       J1 = 0.0 deg, J2 = 0.0 deg
 };
P[142] {
    GP1:
        UF : 6, UT : 5,     CONFIG: 'N U T, 0, 0, 0',
       X = -379.5 mm, Y = 409.2 mm, Z = 657.7 mm,
       W = -12.0 deg, P = 10.7 deg,
    GP2:
        UF : 1, UT : 2,
       J1 = 0.0 deg, J2 = 0.0 deg
 };
P[387] {
    GP1:
        UF : 6, UT : 5,     CONFIG: 'N U T, 0, 0, 0',
 X = -362.5 mm, Y = 480.2 mm, Z = 657.7 mm,       W = -12.0 deg, P = 10.7 deg,
    GP2:
        UF : 1, UT : 2,
       J1 = 0.0 deg, J2 = 0.0 deg
 };
P[143] {
    GP1:
        UF : 6, UT : 5,     CONFIG: 'N U T, 0, 0, 0',
       X = -383.8 mm, Y = 412.9 mm, Z = 657.7 mm,
       W = -11.8 deg, P = 10.5 deg,
    GP2:
        UF : 1, UT : 2,
       J1 = 0.0 deg, J2 = 0.0 deg
 };
P[388] {
    GP1:
        UF : 6, UT : 5,     CONFIG: 'N U T, 0, 0, 0',
 X = -366.8 mm, Y = 483.9 mm, Z = 657.7 mm,       W = -11.8 deg, P = 10.5 deg,
    GP2:
        UF : 1, UT : 2,
       J1 = 0.0 deg, J2 = 0.0 deg
 };
P[144] {
    GP1:
        UF : 6, UT : 5,     CONFIG: 'N U T, 0, 0, 0',
       X = -385.4 mm, Y = 414.3 mm, Z = 657.7 mm,
       W = -12.1 deg, P = 10.1 deg,
    GP2:
        UF : 1, UT : 2,
       J1 = 0.0 deg, J2 = 0.0 deg
 };
P[389] {
    GP1:
        UF : 6, UT : 5,     CONFIG: 'N U T, 0, 0, 0',
 X = -368.4 mm, Y = 485.3 mm, Z = 657.7 mm,       W = -12.1 deg, P = 10.1 deg,
    GP2:
        UF : 1, UT : 2,
       J1 = 0.0 deg, J2 = 0.0 deg
 };
P[145] {
    GP1:
        UF : 6, UT : 5,     CONFIG: 'N U T, 0, 0, 0',
       X = -393.1 mm, Y = 420.6 mm, Z = 657.7 mm,
       W = -12.1 deg, P = 9.4 deg,
    GP2:
        UF : 1, UT : 2,
       J1 = 0.0 deg, J2 = 0.0 deg
 };
P[390] {
    GP1:
        UF : 6, UT : 5,     CONFIG: 'N U T, 0, 0, 0',
 X = -376.1 mm, Y = 491.6 mm, Z = 657.7 mm,       W = -12.1 deg, P = 9.4 deg,
    GP2:
        UF : 1, UT : 2,
       J1 = 0.0 deg, J2 = 0.0 deg
 };
P[146] {
    GP1:
        UF : 6, UT : 5,     CONFIG: 'N U T, 0, 0, 0',
       X = -395.3 mm, Y = 422.2 mm, Z = 657.7 mm,
       W = -12.2 deg, P = 9.4 deg,
    GP2:
        UF : 1, UT : 2,
       J1 = 0.0 deg, J2 = 0.0 deg
 };
P[391] {
    GP1:
        UF : 6, UT : 5,     CONFIG: 'N U T, 0, 0, 0',
 X = -378.3 mm, Y = 493.2 mm, Z = 657.7 mm,       W = -12.2 deg, P = 9.4 deg,
    GP2:
        UF : 1, UT : 2,
       J1 = 0.0 deg, J2 = 0.0 deg
 };
P[147] {
    GP1:
        UF : 6, UT : 5,     CONFIG: 'N U T, 0, 0, 0',
       X = -398.9 mm, Y = 425.0 mm, Z = 657.7 mm,
       W = -12.2 deg, P = 9.5 deg,
    GP2:
        UF : 1, UT : 2,
       J1 = 0.0 deg, J2 = 0.0 deg
 };
P[392] {
    GP1:
        UF : 6, UT : 5,     CONFIG: 'N U T, 0, 0, 0',
 X = -381.9 mm, Y = 496.0 mm, Z = 657.7 mm,       W = -12.2 deg, P = 9.5 deg,
    GP2:
        UF : 1, UT : 2,
       J1 = 0.0 deg, J2 = 0.0 deg
 };
P[148] {
    GP1:
        UF : 6, UT : 5,     CONFIG: 'N U T, 0, 0, 0',
       X = -400.6 mm, Y = 426.4 mm, Z = 657.7 mm,
       W = -11.7 deg, P = 10.2 deg,
    GP2:
        UF : 1, UT : 2,
       J1 = 0.0 deg, J2 = 0.0 deg
 };
P[393] {
    GP1:
        UF : 6, UT : 5,     CONFIG: 'N U T, 0, 0, 0',
 X = -383.6 mm, Y = 497.4 mm, Z = 657.7 mm,       W = -11.7 deg, P = 10.2 deg,
    GP2:
        UF : 1, UT : 2,
       J1 = 0.0 deg, J2 = 0.0 deg
 };
P[149] {
    GP1:
        UF : 6, UT : 5,     CONFIG: 'N U T, 0, 0, 0',
       X = -401.3 mm, Y = 427.0 mm, Z = 657.7 mm,
       W = -11.3 deg, P = 10.7 deg,
    GP2:
        UF : 1, UT : 2,
       J1 = 0.0 deg, J2 = 0.0 deg
 };
P[394] {
    GP1:
        UF : 6, UT : 5,     CONFIG: 'N U T, 0, 0, 0',
 X = -384.3 mm, Y = 498.0 mm, Z = 657.7 mm,       W = -11.3 deg, P = 10.7 deg,
    GP2:
        UF : 1, UT : 2,
       J1 = 0.0 deg, J2 = 0.0 deg
 };
P[150] {
    GP1:
        UF : 6, UT : 5,     CONFIG: 'N U T, 0, 0, 0',
       X = -401.5 mm, Y = 427.2 mm, Z = 657.7 mm,
       W = -11.0 deg, P = 11.0 deg,
    GP2:
        UF : 1, UT : 2,
       J1 = 0.0 deg, J2 = 0.0 deg
 };
P[395] {
    GP1:
        UF : 6, UT : 5,     CONFIG: 'N U T, 0, 0, 0',
 X = -384.5 mm, Y = 498.2 mm, Z = 657.7 mm,       W = -11.0 deg, P = 11.0 deg,
    GP2:
        UF : 1, UT : 2,
       J1 = 0.0 deg, J2 = 0.0 deg
 };
P[151] {
    GP1:
        UF : 6, UT : 5,     CONFIG: 'N U T, 0, 0, 0',
       X = -401.7 mm, Y = 427.4 mm, Z = 657.7 mm,
       W = -10.8 deg, P = 11.3 deg,
    GP2:
        UF : 1, UT : 2,
       J1 = 0.0 deg, J2 = 0.0 deg
 };
P[396] {
    GP1:
        UF : 6, UT : 5,     CONFIG: 'N U T, 0, 0, 0',
 X = -384.7 mm, Y = 498.4 mm, Z = 657.7 mm,       W = -10.8 deg, P = 11.3 deg,
    GP2:
        UF : 1, UT : 2,
       J1 = 0.0 deg, J2 = 0.0 deg
 };
P[152] {
    GP1:
        UF : 6, UT : 5,     CONFIG: 'N U T, 0, 0, 0',
       X = -401.8 mm, Y = 427.6 mm, Z = 657.7 mm,
       W = -10.6 deg, P = 11.6 deg,
    GP2:
        UF : 1, UT : 2,
       J1 = 0.0 deg, J2 = 0.0 deg
 };
P[397] {
    GP1:
        UF : 6, UT : 5,     CONFIG: 'N U T, 0, 0, 0',
 X = -384.8 mm, Y = 498.6 mm, Z = 657.7 mm,       W = -10.6 deg, P = 11.6 deg,
    GP2:
        UF : 1, UT : 2,
       J1 = 0.0 deg, J2 = 0.0 deg
 };
P[153] {
    GP1:
        UF : 6, UT : 5,     CONFIG: 'N U T, 0, 0, 0',
       X = -402.0 mm, Y = 427.7 mm, Z = 657.7 mm,
       W = -10.4 deg, P = 11.9 deg,
    GP2:
        UF : 1, UT : 2,
       J1 = 0.0 deg, J2 = 0.0 deg
 };
P[398] {
    GP1:
        UF : 6, UT : 5,     CONFIG: 'N U T, 0, 0, 0',
 X = -385.0 mm, Y = 498.7 mm, Z = 657.7 mm,       W = -10.4 deg, P = 11.9 deg,
    GP2:
        UF : 1, UT : 2,
       J1 = 0.0 deg, J2 = 0.0 deg
 };
P[154] {
    GP1:
        UF : 6, UT : 5,     CONFIG: 'N U T, 0, 0, 0',
       X = -402.6 mm, Y = 428.5 mm, Z = 657.7 mm,
       W = -10.1 deg, P = 12.4 deg,
    GP2:
        UF : 1, UT : 2,
       J1 = 0.0 deg, J2 = 0.0 deg
 };
P[399] {
    GP1:
        UF : 6, UT : 5,     CONFIG: 'N U T, 0, 0, 0',
 X = -385.6 mm, Y = 499.5 mm, Z = 657.7 mm,       W = -10.1 deg, P = 12.4 deg,
    GP2:
        UF : 1, UT : 2,
       J1 = 0.0 deg, J2 = 0.0 deg
 };
P[155] {
    GP1:
        UF : 6, UT : 5,     CONFIG: 'N U T, 0, 0, 0',
       X = -403.4 mm, Y = 429.5 mm, Z = 657.7 mm,
       W = -9.6 deg, P = 12.8 deg,
    GP2:
        UF : 1, UT : 2,
       J1 = 0.0 deg, J2 = 0.0 deg
 };
P[400] {
    GP1:
        UF : 6, UT : 5,     CONFIG: 'N U T, 0, 0, 0',
 X = -386.4 mm, Y = 500.5 mm, Z = 657.7 mm,       W = -9.6 deg, P = 12.8 deg,
    GP2:
        UF : 1, UT : 2,
       J1 = 0.0 deg, J2 = 0.0 deg
 };
P[156] {
    GP1:
        UF : 6, UT : 5,     CONFIG: 'N U T, 0, 0, 0',
       X = -403.6 mm, Y = 429.7 mm, Z = 657.7 mm,
       W = -9.3 deg, P = 13.0 deg,
    GP2:
        UF : 1, UT : 2,
       J1 = 0.0 deg, J2 = 0.0 deg
 };
P[401] {
    GP1:
        UF : 6, UT : 5,     CONFIG: 'N U T, 0, 0, 0',
 X = -386.6 mm, Y = 500.7 mm, Z = 657.7 mm,       W = -9.3 deg, P = 13.0 deg,
    GP2:
        UF : 1, UT : 2,
       J1 = 0.0 deg, J2 = 0.0 deg
 };
P[157] {
    GP1:
        UF : 6, UT : 5,     CONFIG: 'N U T, 0, 0, 0',
       X = -403.7 mm, Y = 429.9 mm, Z = 657.7 mm,
       W = -9.0 deg, P = 13.2 deg,
    GP2:
        UF : 1, UT : 2,
       J1 = 0.0 deg, J2 = 0.0 deg
 };
P[402] {
    GP1:
        UF : 6, UT : 5,     CONFIG: 'N U T, 0, 0, 0',
 X = -386.7 mm, Y = 500.9 mm, Z = 657.7 mm,       W = -9.0 deg, P = 13.2 deg,
    GP2:
        UF : 1, UT : 2,
       J1 = 0.0 deg, J2 = 0.0 deg
 };
P[158] {
    GP1:
        UF : 6, UT : 5,     CONFIG: 'N U T, 0, 0, 0',
       X = -403.8 mm, Y = 430.1 mm, Z = 657.7 mm,
       W = -8.7 deg, P = 13.4 deg,
    GP2:
        UF : 1, UT : 2,
       J1 = 0.0 deg, J2 = 0.0 deg
 };
P[403] {
    GP1:
        UF : 6, UT : 5,     CONFIG: 'N U T, 0, 0, 0',
 X = -386.8 mm, Y = 501.1 mm, Z = 657.7 mm,       W = -8.7 deg, P = 13.4 deg,
    GP2:
        UF : 1, UT : 2,
       J1 = 0.0 deg, J2 = 0.0 deg
 };
P[159] {
    GP1:
        UF : 6, UT : 5,     CONFIG: 'N U T, 0, 0, 0',
       X = -404.0 mm, Y = 430.3 mm, Z = 657.7 mm,
       W = -8.5 deg, P = 13.6 deg,
    GP2:
        UF : 1, UT : 2,
       J1 = 0.0 deg, J2 = 0.0 deg
 };
P[404] {
    GP1:
        UF : 6, UT : 5,     CONFIG: 'N U T, 0, 0, 0',
 X = -387.0 mm, Y = 501.3 mm, Z = 657.7 mm,       W = -8.5 deg, P = 13.6 deg,
    GP2:
        UF : 1, UT : 2,
       J1 = 0.0 deg, J2 = 0.0 deg
 };
P[160] {
    GP1:
        UF : 6, UT : 5,     CONFIG: 'N U T, 0, 0, 0',
       X = -404.5 mm, Y = 431.2 mm, Z = 657.7 mm,
       W = -7.9 deg, P = 13.8 deg,
    GP2:
        UF : 1, UT : 2,
       J1 = 0.0 deg, J2 = 0.0 deg
 };
P[405] {
    GP1:
        UF : 6, UT : 5,     CONFIG: 'N U T, 0, 0, 0',
 X = -387.5 mm, Y = 502.2 mm, Z = 657.7 mm,       W = -7.9 deg, P = 13.8 deg,
    GP2:
        UF : 1, UT : 2,
       J1 = 0.0 deg, J2 = 0.0 deg
 };
P[161] {
    GP1:
        UF : 6, UT : 5,     CONFIG: 'N U T, 0, 0, 0',
       X = -405.0 mm, Y = 432.1 mm, Z = 657.7 mm,
       W = -7.5 deg, P = 14.1 deg,
    GP2:
        UF : 1, UT : 2,
       J1 = 0.0 deg, J2 = 0.0 deg
 };
P[406] {
    GP1:
        UF : 6, UT : 5,     CONFIG: 'N U T, 0, 0, 0',
 X = -388.0 mm, Y = 503.1 mm, Z = 657.7 mm,       W = -7.5 deg, P = 14.1 deg,
    GP2:
        UF : 1, UT : 2,
       J1 = 0.0 deg, J2 = 0.0 deg
 };
P[162] {
    GP1:
        UF : 6, UT : 5,     CONFIG: 'N U T, 0, 0, 0',
       X = -405.3 mm, Y = 432.7 mm, Z = 657.7 mm,
       W = -6.6 deg, P = 14.4 deg,
    GP2:
        UF : 1, UT : 2,
       J1 = 0.0 deg, J2 = 0.0 deg
 };
P[407] {
    GP1:
        UF : 6, UT : 5,     CONFIG: 'N U T, 0, 0, 0',
 X = -388.3 mm, Y = 503.7 mm, Z = 657.7 mm,       W = -6.6 deg, P = 14.4 deg,
    GP2:
        UF : 1, UT : 2,
       J1 = 0.0 deg, J2 = 0.0 deg
 };
P[163] {
    GP1:
        UF : 6, UT : 5,     CONFIG: 'N U T, 0, 0, 0',
       X = -405.5 mm, Y = 433.2 mm, Z = 657.7 mm,
       W = -5.8 deg, P = 14.6 deg,
    GP2:
        UF : 1, UT : 2,
       J1 = 0.0 deg, J2 = 0.0 deg
 };
P[408] {
    GP1:
        UF : 6, UT : 5,     CONFIG: 'N U T, 0, 0, 0',
 X = -388.5 mm, Y = 504.2 mm, Z = 657.7 mm,       W = -5.8 deg, P = 14.6 deg,
    GP2:
        UF : 1, UT : 2,
       J1 = 0.0 deg, J2 = 0.0 deg
 };
P[164] {
    GP1:
        UF : 6, UT : 5,     CONFIG: 'N U T, 0, 0, 0',
       X = -405.9 mm, Y = 434.5 mm, Z = 657.7 mm,
       W = -5.1 deg, P = 14.6 deg,
    GP2:
        UF : 1, UT : 2,
       J1 = 0.0 deg, J2 = 0.0 deg
 };
P[409] {
    GP1:
        UF : 6, UT : 5,     CONFIG: 'N U T, 0, 0, 0',
 X = -388.9 mm, Y = 505.5 mm, Z = 657.7 mm,       W = -5.1 deg, P = 14.6 deg,
    GP2:
        UF : 1, UT : 2,
       J1 = 0.0 deg, J2 = 0.0 deg
 };
P[165] {
    GP1:
        UF : 6, UT : 5,     CONFIG: 'N U T, 0, 0, 0',
       X = -406.2 mm, Y = 435.2 mm, Z = 657.7 mm,
       W = -4.6 deg, P = 14.8 deg,
    GP2:
        UF : 1, UT : 2,
       J1 = 0.0 deg, J2 = 0.0 deg
 };
P[410] {
    GP1:
        UF : 6, UT : 5,     CONFIG: 'N U T, 0, 0, 0',
 X = -389.2 mm, Y = 506.2 mm, Z = 657.7 mm,       W = -4.6 deg, P = 14.8 deg,
    GP2:
        UF : 1, UT : 2,
       J1 = 0.0 deg, J2 = 0.0 deg
 };
P[166] {
    GP1:
        UF : 6, UT : 5,     CONFIG: 'N U T, 0, 0, 0',
       X = -406.4 mm, Y = 435.8 mm, Z = 657.7 mm,
       W = -3.7 deg, P = 14.9 deg,
    GP2:
        UF : 1, UT : 2,
       J1 = 0.0 deg, J2 = 0.0 deg
 };
P[411] {
    GP1:
        UF : 6, UT : 5,     CONFIG: 'N U T, 0, 0, 0',
 X = -389.4 mm, Y = 506.8 mm, Z = 657.7 mm,       W = -3.7 deg, P = 14.9 deg,
    GP2:
        UF : 1, UT : 2,
       J1 = 0.0 deg, J2 = 0.0 deg
 };
P[167] {
    GP1:
        UF : 6, UT : 5,     CONFIG: 'N U T, 0, 0, 0',
       X = -406.5 mm, Y = 436.4 mm, Z = 657.7 mm,
       W = -2.8 deg, P = 14.7 deg,
    GP2:
        UF : 1, UT : 2,
       J1 = 0.0 deg, J2 = 0.0 deg
 };
P[412] {
    GP1:
        UF : 6, UT : 5,     CONFIG: 'N U T, 0, 0, 0',
 X = -389.5 mm, Y = 507.4 mm, Z = 657.7 mm,       W = -2.8 deg, P = 14.7 deg,
    GP2:
        UF : 1, UT : 2,
       J1 = 0.0 deg, J2 = 0.0 deg
 };
P[168] {
    GP1:
        UF : 6, UT : 5,     CONFIG: 'N U T, 0, 0, 0',
       X = -406.7 mm, Y = 437.8 mm, Z = 657.7 mm,
       W = -2.2 deg, P = 14.0 deg,
    GP2:
        UF : 1, UT : 2,
       J1 = 0.0 deg, J2 = 0.0 deg
 };
P[413] {
    GP1:
        UF : 6, UT : 5,     CONFIG: 'N U T, 0, 0, 0',
 X = -389.7 mm, Y = 508.8 mm, Z = 657.7 mm,       W = -2.2 deg, P = 14.0 deg,
    GP2:
        UF : 1, UT : 2,
       J1 = 0.0 deg, J2 = 0.0 deg
 };
P[169] {
    GP1:
        UF : 6, UT : 5,     CONFIG: 'N U T, 0, 0, 0',
       X = -406.8 mm, Y = 438.6 mm, Z = 657.7 mm,
       W = -1.3 deg, P = 13.5 deg,
    GP2:
        UF : 1, UT : 2,
       J1 = 0.0 deg, J2 = 0.0 deg
 };
P[414] {
    GP1:
        UF : 6, UT : 5,     CONFIG: 'N U T, 0, 0, 0',
 X = -389.8 mm, Y = 509.6 mm, Z = 657.7 mm,       W = -1.3 deg, P = 13.5 deg,
    GP2:
        UF : 1, UT : 2,
       J1 = 0.0 deg, J2 = 0.0 deg
 };
P[170] {
    GP1:
        UF : 6, UT : 5,     CONFIG: 'N U T, 0, 0, 0',
       X = -406.9 mm, Y = 439.5 mm, Z = 657.7 mm,
       W = -0.4 deg, P = 13.3 deg,
    GP2:
        UF : 1, UT : 2,
       J1 = 0.0 deg, J2 = 0.0 deg
 };
P[415] {
    GP1:
        UF : 6, UT : 5,     CONFIG: 'N U T, 0, 0, 0',
 X = -389.9 mm, Y = 510.5 mm, Z = 657.7 mm,       W = -0.4 deg, P = 13.3 deg,
    GP2:
        UF : 1, UT : 2,
       J1 = 0.0 deg, J2 = 0.0 deg
 };
P[171] {
    GP1:
        UF : 6, UT : 5,     CONFIG: 'N U T, 0, 0, 0',
       X = -406.9 mm, Y = 440.5 mm, Z = 657.7 mm,
       W = 0.2 deg, P = 13.1 deg,
    GP2:
        UF : 1, UT : 2,
       J1 = 0.0 deg, J2 = 0.0 deg
 };
P[416] {
    GP1:
        UF : 6, UT : 5,     CONFIG: 'N U T, 0, 0, 0',
 X = -389.9 mm, Y = 511.5 mm, Z = 657.7 mm,       W = 0.2 deg, P = 13.1 deg,
    GP2:
        UF : 1, UT : 2,
       J1 = 0.0 deg, J2 = 0.0 deg
 };
P[172] {
    GP1:
        UF : 6, UT : 5,     CONFIG: 'N U T, 0, 0, 0',
       X = -406.8 mm, Y = 441.6 mm, Z = 657.7 mm,
       W = 0.9 deg, P = 12.6 deg,
    GP2:
        UF : 1, UT : 2,
       J1 = 0.0 deg, J2 = 0.0 deg
 };
P[417] {
    GP1:
        UF : 6, UT : 5,     CONFIG: 'N U T, 0, 0, 0',
 X = -389.8 mm, Y = 512.6 mm, Z = 657.7 mm,       W = 0.9 deg, P = 12.6 deg,
    GP2:
        UF : 1, UT : 2,
       J1 = 0.0 deg, J2 = 0.0 deg
 };
P[173] {
    GP1:
        UF : 6, UT : 5,     CONFIG: 'N U T, 0, 0, 0',
       X = -406.8 mm, Y = 441.8 mm, Z = 657.7 mm,
       W = 1.2 deg, P = 12.4 deg,
    GP2:
        UF : 1, UT : 2,
       J1 = 0.0 deg, J2 = 0.0 deg
 };
P[418] {
    GP1:
        UF : 6, UT : 5,     CONFIG: 'N U T, 0, 0, 0',
 X = -389.8 mm, Y = 512.8 mm, Z = 657.7 mm,       W = 1.2 deg, P = 12.4 deg,
    GP2:
        UF : 1, UT : 2,
       J1 = 0.0 deg, J2 = 0.0 deg
 };
P[174] {
    GP1:
        UF : 6, UT : 5,     CONFIG: 'N U T, 0, 0, 0',
       X = -406.8 mm, Y = 442.1 mm, Z = 657.7 mm,
       W = 1.4 deg, P = 12.2 deg,
    GP2:
        UF : 1, UT : 2,
       J1 = 0.0 deg, J2 = 0.0 deg
 };
P[419] {
    GP1:
        UF : 6, UT : 5,     CONFIG: 'N U T, 0, 0, 0',
 X = -389.8 mm, Y = 513.1 mm, Z = 657.7 mm,       W = 1.4 deg, P = 12.2 deg,
    GP2:
        UF : 1, UT : 2,
       J1 = 0.0 deg, J2 = 0.0 deg
 };
P[175] {
    GP1:
        UF : 6, UT : 5,     CONFIG: 'N U T, 0, 0, 0',
       X = -406.8 mm, Y = 442.4 mm, Z = 657.7 mm,
       W = 1.7 deg, P = 12.1 deg,
    GP2:
        UF : 1, UT : 2,
       J1 = 0.0 deg, J2 = 0.0 deg
 };
P[420] {
    GP1:
        UF : 6, UT : 5,     CONFIG: 'N U T, 0, 0, 0',
 X = -389.8 mm, Y = 513.4 mm, Z = 657.7 mm,       W = 1.7 deg, P = 12.1 deg,
    GP2:
        UF : 1, UT : 2,
       J1 = 0.0 deg, J2 = 0.0 deg
 };
P[176] {
    GP1:
        UF : 6, UT : 5,     CONFIG: 'N U T, 0, 0, 0',
       X = -406.7 mm, Y = 442.6 mm, Z = 657.7 mm,
       W = 1.9 deg, P = 11.9 deg,
    GP2:
        UF : 1, UT : 2,
       J1 = 0.0 deg, J2 = 0.0 deg
 };
P[421] {
    GP1:
        UF : 6, UT : 5,     CONFIG: 'N U T, 0, 0, 0',
 X = -389.7 mm, Y = 513.6 mm, Z = 657.7 mm,       W = 1.9 deg, P = 11.9 deg,
    GP2:
        UF : 1, UT : 2,
       J1 = 0.0 deg, J2 = 0.0 deg
 };
P[177] {
    GP1:
        UF : 6, UT : 5,     CONFIG: 'N U T, 0, 0, 0',
       X = -406.4 mm, Y = 444.4 mm, Z = 657.7 mm,
       W = 2.3 deg, P = 10.3 deg,
    GP2:
        UF : 1, UT : 2,
       J1 = 0.0 deg, J2 = 0.0 deg
 };
P[422] {
    GP1:
        UF : 6, UT : 5,     CONFIG: 'N U T, 0, 0, 0',
 X = -389.4 mm, Y = 515.4 mm, Z = 657.7 mm,       W = 2.3 deg, P = 10.3 deg,
    GP2:
        UF : 1, UT : 2,
       J1 = 0.0 deg, J2 = 0.0 deg
 };
P[178] {
    GP1:
        UF : 6, UT : 5,     CONFIG: 'N U T, 0, 0, 0',
       X = -406.2 mm, Y = 445.1 mm, Z = 657.7 mm,
       W = 2.7 deg, P = 9.6 deg,
    GP2:
        UF : 1, UT : 2,
       J1 = 0.0 deg, J2 = 0.0 deg
 };
P[423] {
    GP1:
        UF : 6, UT : 5,     CONFIG: 'N U T, 0, 0, 0',
 X = -389.2 mm, Y = 516.1 mm, Z = 657.7 mm,       W = 2.7 deg, P = 9.6 deg,
    GP2:
        UF : 1, UT : 2,
       J1 = 0.0 deg, J2 = 0.0 deg
 };
P[179] {
    GP1:
        UF : 6, UT : 5,     CONFIG: 'N U T, 0, 0, 0',
       X = -406.0 mm, Y = 445.9 mm, Z = 657.7 mm,
       W = 3.2 deg, P = 9.1 deg,
    GP2:
        UF : 1, UT : 2,
       J1 = 0.0 deg, J2 = 0.0 deg
 };
P[424] {
    GP1:
        UF : 6, UT : 5,     CONFIG: 'N U T, 0, 0, 0',
 X = -389.0 mm, Y = 516.9 mm, Z = 657.7 mm,       W = 3.2 deg, P = 9.1 deg,
    GP2:
        UF : 1, UT : 2,
       J1 = 0.0 deg, J2 = 0.0 deg
 };
P[180] {
    GP1:
        UF : 6, UT : 5,     CONFIG: 'N U T, 0, 0, 0',
       X = -405.6 mm, Y = 446.9 mm, Z = 657.7 mm,
       W = 3.4 deg, P = 8.9 deg,
    GP2:
        UF : 1, UT : 2,
       J1 = 0.0 deg, J2 = 0.0 deg
 };
P[425] {
    GP1:
        UF : 6, UT : 5,     CONFIG: 'N U T, 0, 0, 0',
 X = -388.6 mm, Y = 517.9 mm, Z = 657.7 mm,       W = 3.4 deg, P = 8.9 deg,
    GP2:
        UF : 1, UT : 2,
       J1 = 0.0 deg, J2 = 0.0 deg
 };
P[181] {
    GP1:
        UF : 6, UT : 5,     CONFIG: 'N U T, 0, 0, 0',
       X = -405.4 mm, Y = 447.3 mm, Z = 657.7 mm,
       W = 3.7 deg, P = 8.6 deg,
    GP2:
        UF : 1, UT : 2,
       J1 = 0.0 deg, J2 = 0.0 deg
 };
P[426] {
    GP1:
        UF : 6, UT : 5,     CONFIG: 'N U T, 0, 0, 0',
 X = -388.4 mm, Y = 518.3 mm, Z = 657.7 mm,       W = 3.7 deg, P = 8.6 deg,
    GP2:
        UF : 1, UT : 2,
       J1 = 0.0 deg, J2 = 0.0 deg
 };
P[182] {
    GP1:
        UF : 6, UT : 5,     CONFIG: 'N U T, 0, 0, 0',
       X = -405.3 mm, Y = 447.5 mm, Z = 657.7 mm,
       W = 3.8 deg, P = 8.4 deg,
    GP2:
        UF : 1, UT : 2,
       J1 = 0.0 deg, J2 = 0.0 deg
 };
P[427] {
    GP1:
        UF : 6, UT : 5,     CONFIG: 'N U T, 0, 0, 0',
 X = -388.3 mm, Y = 518.5 mm, Z = 657.7 mm,       W = 3.8 deg, P = 8.4 deg,
    GP2:
        UF : 1, UT : 2,
       J1 = 0.0 deg, J2 = 0.0 deg
 };
P[183] {
    GP1:
        UF : 6, UT : 5,     CONFIG: 'N U T, 0, 0, 0',
       X = -405.2 mm, Y = 447.7 mm, Z = 657.7 mm,
       W = 3.9 deg, P = 8.2 deg,
    GP2:
        UF : 1, UT : 2,
       J1 = 0.0 deg, J2 = 0.0 deg
 };
P[428] {
    GP1:
        UF : 6, UT : 5,     CONFIG: 'N U T, 0, 0, 0',
 X = -388.2 mm, Y = 518.7 mm, Z = 657.7 mm,       W = 3.9 deg, P = 8.2 deg,
    GP2:
        UF : 1, UT : 2,
       J1 = 0.0 deg, J2 = 0.0 deg
 };
P[184] {
    GP1:
        UF : 6, UT : 5,     CONFIG: 'N U T, 0, 0, 0',
       X = -404.8 mm, Y = 448.5 mm, Z = 657.7 mm,
       W = 3.8 deg, P = 7.1 deg,
    GP2:
        UF : 1, UT : 2,
       J1 = 0.0 deg, J2 = 0.0 deg
 };
P[429] {
    GP1:
        UF : 6, UT : 5,     CONFIG: 'N U T, 0, 0, 0',
 X = -387.8 mm, Y = 519.5 mm, Z = 657.7 mm,       W = 3.8 deg, P = 7.1 deg,
    GP2:
        UF : 1, UT : 2,
       J1 = 0.0 deg, J2 = 0.0 deg
 };
P[185] {
    GP1:
        UF : 6, UT : 5,     CONFIG: 'N U T, 0, 0, 0',
       X = -404.1 mm, Y = 449.8 mm, Z = 657.7 mm,
       W = 3.6 deg, P = 6.2 deg,
    GP2:
        UF : 1, UT : 2,
       J1 = 0.0 deg, J2 = 0.0 deg
 };
P[430] {
    GP1:
        UF : 6, UT : 5,     CONFIG: 'N U T, 0, 0, 0',
 X = -387.1 mm, Y = 520.8 mm, Z = 657.7 mm,       W = 3.6 deg, P = 6.2 deg,
    GP2:
        UF : 1, UT : 2,
       J1 = 0.0 deg, J2 = 0.0 deg
 };
P[186] {
    GP1:
        UF : 6, UT : 5,     CONFIG: 'N U T, 0, 0, 0',
       X = -404.0 mm, Y = 450.0 mm, Z = 657.7 mm,
       W = 3.6 deg, P = 6.0 deg,
    GP2:
        UF : 1, UT : 2,
       J1 = 0.0 deg, J2 = 0.0 deg
 };
P[431] {
    GP1:
        UF : 6, UT : 5,     CONFIG: 'N U T, 0, 0, 0',
 X = -387.0 mm, Y = 521.0 mm, Z = 657.7 mm,       W = 3.6 deg, P = 6.0 deg,
    GP2:
        UF : 1, UT : 2,
       J1 = 0.0 deg, J2 = 0.0 deg
 };
P[187] {
    GP1:
        UF : 6, UT : 5,     CONFIG: 'N U T, 0, 0, 0',
       X = -403.9 mm, Y = 450.2 mm, Z = 657.7 mm,
       W = 3.7 deg, P = 5.8 deg,
    GP2:
        UF : 1, UT : 2,
       J1 = 0.0 deg, J2 = 0.0 deg
 };
P[432] {
    GP1:
        UF : 6, UT : 5,     CONFIG: 'N U T, 0, 0, 0',
 X = -386.9 mm, Y = 521.2 mm, Z = 657.7 mm,       W = 3.7 deg, P = 5.8 deg,
    GP2:
        UF : 1, UT : 2,
       J1 = 0.0 deg, J2 = 0.0 deg
 };
P[188] {
    GP1:
        UF : 6, UT : 5,     CONFIG: 'N U T, 0, 0, 0',
       X = -403.8 mm, Y = 450.4 mm, Z = 657.7 mm,
       W = 3.7 deg, P = 5.6 deg,
    GP2:
        UF : 1, UT : 2,
       J1 = 0.0 deg, J2 = 0.0 deg
 };
P[433] {
    GP1:
        UF : 6, UT : 5,     CONFIG: 'N U T, 0, 0, 0',
 X = -386.8 mm, Y = 521.4 mm, Z = 657.7 mm,       W = 3.7 deg, P = 5.6 deg,
    GP2:
        UF : 1, UT : 2,
       J1 = 0.0 deg, J2 = 0.0 deg
 };
P[189] {
    GP1:
        UF : 6, UT : 5,     CONFIG: 'N U T, 0, 0, 0',
       X = -403.6 mm, Y = 450.6 mm, Z = 657.7 mm,
       W = 3.8 deg, P = 5.4 deg,
    GP2:
        UF : 1, UT : 2,
       J1 = 0.0 deg, J2 = 0.0 deg
 };
P[434] {
    GP1:
        UF : 6, UT : 5,     CONFIG: 'N U T, 0, 0, 0',
 X = -386.6 mm, Y = 521.6 mm, Z = 657.7 mm,       W = 3.8 deg, P = 5.4 deg,
    GP2:
        UF : 1, UT : 2,
       J1 = 0.0 deg, J2 = 0.0 deg
 };
P[190] {
    GP1:
        UF : 6, UT : 5,     CONFIG: 'N U T, 0, 0, 0',
       X = -403.3 mm, Y = 451.0 mm, Z = 657.7 mm,
       W = 3.6 deg, P = 4.7 deg,
    GP2:
        UF : 1, UT : 2,
       J1 = 0.0 deg, J2 = 0.0 deg
 };
P[435] {
    GP1:
        UF : 6, UT : 5,     CONFIG: 'N U T, 0, 0, 0',
 X = -386.3 mm, Y = 522.0 mm, Z = 657.7 mm,       W = 3.6 deg, P = 4.7 deg,
    GP2:
        UF : 1, UT : 2,
       J1 = 0.0 deg, J2 = 0.0 deg
 };
P[191] {
    GP1:
        UF : 6, UT : 5,     CONFIG: 'N U T, 0, 0, 0',
       X = -403.1 mm, Y = 451.2 mm, Z = 657.7 mm,
       W = 3.5 deg, P = 4.4 deg,
    GP2:
        UF : 1, UT : 2,
       J1 = 0.0 deg, J2 = 0.0 deg
 };
P[436] {
    GP1:
        UF : 6, UT : 5,     CONFIG: 'N U T, 0, 0, 0',
 X = -386.1 mm, Y = 522.2 mm, Z = 657.7 mm,       W = 3.5 deg, P = 4.4 deg,
    GP2:
        UF : 1, UT : 2,
       J1 = 0.0 deg, J2 = 0.0 deg
 };
P[192] {
    GP1:
        UF : 6, UT : 5,     CONFIG: 'N U T, 0, 0, 0',
       X = -403.0 mm, Y = 451.5 mm, Z = 657.7 mm,
       W = 3.3 deg, P = 4.1 deg,
    GP2:
        UF : 1, UT : 2,
       J1 = 0.0 deg, J2 = 0.0 deg
 };
P[437] {
    GP1:
        UF : 6, UT : 5,     CONFIG: 'N U T, 0, 0, 0',
 X = -386.0 mm, Y = 522.5 mm, Z = 657.7 mm,       W = 3.3 deg, P = 4.1 deg,
    GP2:
        UF : 1, UT : 2,
       J1 = 0.0 deg, J2 = 0.0 deg
 };
P[193] {
    GP1:
        UF : 6, UT : 5,     CONFIG: 'N U T, 0, 0, 0',
       X = -402.1 mm, Y = 452.5 mm, Z = 657.7 mm,
       W = 3.0 deg, P = 3.6 deg,
    GP2:
        UF : 1, UT : 2,
       J1 = 0.0 deg, J2 = 0.0 deg
 };
P[438] {
    GP1:
        UF : 6, UT : 5,     CONFIG: 'N U T, 0, 0, 0',
 X = -385.1 mm, Y = 523.5 mm, Z = 657.7 mm,       W = 3.0 deg, P = 3.6 deg,
    GP2:
        UF : 1, UT : 2,
       J1 = 0.0 deg, J2 = 0.0 deg
 };
P[194] {
    GP1:
        UF : 6, UT : 5,     CONFIG: 'N U T, 0, 0, 0',
       X = -395.3 mm, Y = 459.8 mm, Z = 657.7 mm,
       W = 2.8 deg, P = 3.4 deg,
    GP2:
        UF : 1, UT : 2,
       J1 = 0.0 deg, J2 = 0.0 deg
 };
P[439] {
    GP1:
        UF : 6, UT : 5,     CONFIG: 'N U T, 0, 0, 0',
 X = -378.3 mm, Y = 530.8 mm, Z = 657.7 mm,       W = 2.8 deg, P = 3.4 deg,
    GP2:
        UF : 1, UT : 2,
       J1 = 0.0 deg, J2 = 0.0 deg
 };
P[195] {
    GP1:
        UF : 6, UT : 5,     CONFIG: 'N U T, 0, 0, 0',
       X = -388.3 mm, Y = 466.9 mm, Z = 657.7 mm,
       W = 2.6 deg, P = 3.2 deg,
    GP2:
        UF : 1, UT : 2,
       J1 = 0.0 deg, J2 = 0.0 deg
 };
P[440] {
    GP1:
        UF : 6, UT : 5,     CONFIG: 'N U T, 0, 0, 0',
 X = -371.3 mm, Y = 537.9 mm, Z = 657.7 mm,       W = 2.6 deg, P = 3.2 deg,
    GP2:
        UF : 1, UT : 2,
       J1 = 0.0 deg, J2 = 0.0 deg
 };
P[196] {
    GP1:
        UF : 6, UT : 5,     CONFIG: 'N U T, 0, 0, 0',
       X = -381.1 mm, Y = 473.9 mm, Z = 657.7 mm,
       W = 2.5 deg, P = 2.9 deg,
    GP2:
        UF : 1, UT : 2,
       J1 = 0.0 deg, J2 = 0.0 deg
 };
P[441] {
    GP1:
        UF : 6, UT : 5,     CONFIG: 'N U T, 0, 0, 0',
 X = -364.1 mm, Y = 544.9 mm, Z = 657.7 mm,       W = 2.5 deg, P = 2.9 deg,
    GP2:
        UF : 1, UT : 2,
       J1 = 0.0 deg, J2 = 0.0 deg
 };
P[197] {
    GP1:
        UF : 6, UT : 5,     CONFIG: 'N U T, 0, 0, 0',
       X = -379.6 mm, Y = 475.3 mm, Z = 657.7 mm,
       W = 2.4 deg, P = 2.9 deg,
    GP2:
        UF : 1, UT : 2,
       J1 = 0.0 deg, J2 = 0.0 deg
 };
P[442] {
    GP1:
        UF : 6, UT : 5,     CONFIG: 'N U T, 0, 0, 0',
 X = -362.6 mm, Y = 546.3 mm, Z = 657.7 mm,       W = 2.4 deg, P = 2.9 deg,
    GP2:
        UF : 1, UT : 2,
       J1 = 0.0 deg, J2 = 0.0 deg
 };
P[198] {
    GP1:
        UF : 6, UT : 5,     CONFIG: 'N U T, 0, 0, 0',
       X = -378.9 mm, Y = 476.2 mm, Z = 657.7 mm,
       W = 2.4 deg, P = 2.9 deg,
    GP2:
        UF : 1, UT : 2,
       J1 = 0.0 deg, J2 = 0.0 deg
 };
P[443] {
    GP1:
        UF : 6, UT : 5,     CONFIG: 'N U T, 0, 0, 0',
 X = -361.9 mm, Y = 547.2 mm, Z = 657.7 mm,       W = 2.4 deg, P = 2.9 deg,
    GP2:
        UF : 1, UT : 2,
       J1 = 0.0 deg, J2 = 0.0 deg
 };
P[199] {
    GP1:
        UF : 6, UT : 5,     CONFIG: 'N U T, 0, 0, 0',
       X = -378.1 mm, Y = 477.2 mm, Z = 657.7 mm,
       W = 2.4 deg, P = 2.8 deg,
    GP2:
        UF : 1, UT : 2,
       J1 = 0.0 deg, J2 = 0.0 deg
 };
P[444] {
    GP1:
        UF : 6, UT : 5,     CONFIG: 'N U T, 0, 0, 0',
 X = -361.1 mm, Y = 548.2 mm, Z = 657.7 mm,       W = 2.4 deg, P = 2.8 deg,
    GP2:
        UF : 1, UT : 2,
       J1 = 0.0 deg, J2 = 0.0 deg
 };
P[200] {
    GP1:
        UF : 6, UT : 5,     CONFIG: 'N U T, 0, 0, 0',
       X = -377.5 mm, Y = 478.2 mm, Z = 657.7 mm,
       W = 2.4 deg, P = 2.8 deg,
    GP2:
        UF : 1, UT : 2,
       J1 = 0.0 deg, J2 = 0.0 deg
 };
P[445] {
    GP1:
        UF : 6, UT : 5,     CONFIG: 'N U T, 0, 0, 0',
 X = -360.5 mm, Y = 549.2 mm, Z = 657.7 mm,       W = 2.4 deg, P = 2.8 deg,
    GP2:
        UF : 1, UT : 2,
       J1 = 0.0 deg, J2 = 0.0 deg
 };
P[201] {
    GP1:
        UF : 6, UT : 5,     CONFIG: 'N U T, 0, 0, 0',
       X = -376.5 mm, Y = 480.4 mm, Z = 657.7 mm,
       W = 2.3 deg, P = 2.8 deg,
    GP2:
        UF : 1, UT : 2,
       J1 = 0.0 deg, J2 = 0.0 deg
 };
P[446] {
    GP1:
        UF : 6, UT : 5,     CONFIG: 'N U T, 0, 0, 0',
 X = -359.5 mm, Y = 551.4 mm, Z = 657.7 mm,       W = 2.3 deg, P = 2.8 deg,
    GP2:
        UF : 1, UT : 2,
       J1 = 0.0 deg, J2 = 0.0 deg
 };
P[202] {
    GP1:
        UF : 6, UT : 5,     CONFIG: 'N U T, 0, 0, 0',
       X = -376.1 mm, Y = 482.5 mm, Z = 657.7 mm,
       W = 2.3 deg, P = 2.7 deg,
    GP2:
        UF : 1, UT : 2,
       J1 = 0.0 deg, J2 = 0.0 deg
 };
P[447] {
    GP1:
        UF : 6, UT : 5,     CONFIG: 'N U T, 0, 0, 0',
 X = -359.1 mm, Y = 553.5 mm, Z = 657.7 mm,       W = 2.3 deg, P = 2.7 deg,
    GP2:
        UF : 1, UT : 2,
       J1 = 0.0 deg, J2 = 0.0 deg
 };
P[203] {
    GP1:
        UF : 6, UT : 5,     CONFIG: 'N U T, 0, 0, 0',
       X = -376.0 mm, Y = 484.4 mm, Z = 657.7 mm,
       W = 2.2 deg, P = 2.7 deg,
    GP2:
        UF : 1, UT : 2,
       J1 = 0.0 deg, J2 = 0.0 deg
 };
P[448] {
    GP1:
        UF : 6, UT : 5,     CONFIG: 'N U T, 0, 0, 0',
 X = -359.0 mm, Y = 555.4 mm, Z = 657.7 mm,       W = 2.2 deg, P = 2.7 deg,
    GP2:
        UF : 1, UT : 2,
       J1 = 0.0 deg, J2 = 0.0 deg
 };
P[204] {
    GP1:
        UF : 6, UT : 5,     CONFIG: 'N U T, 0, 0, 0',
       X = -376.2 mm, Y = 486.0 mm, Z = 657.7 mm,
       W = 2.2 deg, P = 2.6 deg,
    GP2:
        UF : 1, UT : 2,
       J1 = 0.0 deg, J2 = 0.0 deg
 };
P[449] {
    GP1:
        UF : 6, UT : 5,     CONFIG: 'N U T, 0, 0, 0',
 X = -359.2 mm, Y = 557.0 mm, Z = 657.7 mm,       W = 2.2 deg, P = 2.6 deg,
    GP2:
        UF : 1, UT : 2,
       J1 = 0.0 deg, J2 = 0.0 deg
 };
P[205] {
    GP1:
        UF : 6, UT : 5,     CONFIG: 'N U T, 0, 0, 0',
       X = -376.6 mm, Y = 487.6 mm, Z = 657.7 mm,
       W = 2.2 deg, P = 2.6 deg,
    GP2:
        UF : 1, UT : 2,
       J1 = 0.0 deg, J2 = 0.0 deg
 };
P[450] {
    GP1:
        UF : 6, UT : 5,     CONFIG: 'N U T, 0, 0, 0',
 X = -359.6 mm, Y = 558.6 mm, Z = 657.7 mm,       W = 2.2 deg, P = 2.6 deg,
    GP2:
        UF : 1, UT : 2,
       J1 = 0.0 deg, J2 = 0.0 deg
 };
P[206] {
    GP1:
        UF : 6, UT : 5,     CONFIG: 'N U T, 0, 0, 0',
       X = -377.3 mm, Y = 489.3 mm, Z = 657.7 mm,
       W = 2.2 deg, P = 2.6 deg,
    GP2:
        UF : 1, UT : 2,
       J1 = 0.0 deg, J2 = 0.0 deg
 };
P[451] {
    GP1:
        UF : 6, UT : 5,     CONFIG: 'N U T, 0, 0, 0',
 X = -360.3 mm, Y = 560.3 mm, Z = 657.7 mm,       W = 2.2 deg, P = 2.6 deg,
    GP2:
        UF : 1, UT : 2,
       J1 = 0.0 deg, J2 = 0.0 deg
 };
P[207] {
    GP1:
        UF : 6, UT : 5,     CONFIG: 'N U T, 0, 0, 0',
       X = -377.9 mm, Y = 490.3 mm, Z = 657.7 mm,
       W = 2.1 deg, P = 2.5 deg,
    GP2:
        UF : 1, UT : 2,
       J1 = 0.0 deg, J2 = 0.0 deg
 };
P[452] {
    GP1:
        UF : 6, UT : 5,     CONFIG: 'N U T, 0, 0, 0',
 X = -360.9 mm, Y = 561.3 mm, Z = 657.7 mm,       W = 2.1 deg, P = 2.5 deg,
    GP2:
        UF : 1, UT : 2,
       J1 = 0.0 deg, J2 = 0.0 deg
 };
P[208] {
    GP1:
        UF : 6, UT : 5,     CONFIG: 'N U T, 0, 0, 0',
       X = -378.7 mm, Y = 491.3 mm, Z = 657.7 mm,
       W = 2.1 deg, P = 2.5 deg,
    GP2:
        UF : 1, UT : 2,
       J1 = 0.0 deg, J2 = 0.0 deg
 };
P[453] {
    GP1:
        UF : 6, UT : 5,     CONFIG: 'N U T, 0, 0, 0',
 X = -361.7 mm, Y = 562.3 mm, Z = 657.7 mm,       W = 2.1 deg, P = 2.5 deg,
    GP2:
        UF : 1, UT : 2,
       J1 = 0.0 deg, J2 = 0.0 deg
 };
P[209] {
    GP1:
        UF : 6, UT : 5,     CONFIG: 'N U T, 0, 0, 0',
       X = -379.8 mm, Y = 492.3 mm, Z = 657.7 mm,
       W = 2.1 deg, P = 2.5 deg,
    GP2:
        UF : 1, UT : 2,
       J1 = 0.0 deg, J2 = 0.0 deg
 };
P[454] {
    GP1:
        UF : 6, UT : 5,     CONFIG: 'N U T, 0, 0, 0',
 X = -362.8 mm, Y = 563.3 mm, Z = 657.7 mm,       W = 2.1 deg, P = 2.5 deg,
    GP2:
        UF : 1, UT : 2,
       J1 = 0.0 deg, J2 = 0.0 deg
 };
P[210] {
    GP1:
        UF : 6, UT : 5,     CONFIG: 'N U T, 0, 0, 0',
       X = -381.5 mm, Y = 493.5 mm, Z = 657.7 mm,
       W = 2.1 deg, P = 2.4 deg,
    GP2:
        UF : 1, UT : 2,
       J1 = 0.0 deg, J2 = 0.0 deg
 };
P[455] {
    GP1:
        UF : 6, UT : 5,     CONFIG: 'N U T, 0, 0, 0',
 X = -364.5 mm, Y = 564.5 mm, Z = 657.7 mm,       W = 2.1 deg, P = 2.4 deg,
    GP2:
        UF : 1, UT : 2,
       J1 = 0.0 deg, J2 = 0.0 deg
 };
P[211] {
    GP1:
        UF : 6, UT : 5,     CONFIG: 'N U T, 0, 0, 0',
       X = -389.7 mm, Y = 498.8 mm, Z = 657.7 mm,
       W = 1.8 deg, P = 2.2 deg,
    GP2:
        UF : 1, UT : 2,
       J1 = 0.0 deg, J2 = 0.0 deg
 };
P[456] {
    GP1:
        UF : 6, UT : 5,     CONFIG: 'N U T, 0, 0, 0',
 X = -372.7 mm, Y = 569.8 mm, Z = 657.7 mm,       W = 1.8 deg, P = 2.2 deg,
    GP2:
        UF : 1, UT : 2,
       J1 = 0.0 deg, J2 = 0.0 deg
 };
P[212] {
    GP1:
        UF : 6, UT : 5,     CONFIG: 'N U T, 0, 0, 0',
       X = -398.1 mm, Y = 503.9 mm, Z = 657.7 mm,
       W = 1.7 deg, P = 2.0 deg,
    GP2:
        UF : 1, UT : 2,
       J1 = 0.0 deg, J2 = 0.0 deg
 };
P[457] {
    GP1:
        UF : 6, UT : 5,     CONFIG: 'N U T, 0, 0, 0',
 X = -381.1 mm, Y = 574.9 mm, Z = 657.7 mm,       W = 1.7 deg, P = 2.0 deg,
    GP2:
        UF : 1, UT : 2,
       J1 = 0.0 deg, J2 = 0.0 deg
 };
P[213] {
    GP1:
        UF : 6, UT : 5,     CONFIG: 'N U T, 0, 0, 0',
       X = -406.6 mm, Y = 508.9 mm, Z = 657.7 mm,
       W = 1.5 deg, P = 1.8 deg,
    GP2:
        UF : 1, UT : 2,
       J1 = 0.0 deg, J2 = 0.0 deg
 };
P[458] {
    GP1:
        UF : 6, UT : 5,     CONFIG: 'N U T, 0, 0, 0',
 X = -389.6 mm, Y = 579.9 mm, Z = 657.7 mm,       W = 1.5 deg, P = 1.8 deg,
    GP2:
        UF : 1, UT : 2,
       J1 = 0.0 deg, J2 = 0.0 deg
 };
P[214] {
    GP1:
        UF : 6, UT : 5,     CONFIG: 'N U T, 0, 0, 0',
       X = -415.2 mm, Y = 513.7 mm, Z = 657.7 mm,
       W = 1.3 deg, P = 1.5 deg,
    GP2:
        UF : 1, UT : 2,
       J1 = 0.0 deg, J2 = 0.0 deg
 };
P[459] {
    GP1:
        UF : 6, UT : 5,     CONFIG: 'N U T, 0, 0, 0',
 X = -398.2 mm, Y = 584.7 mm, Z = 657.7 mm,       W = 1.3 deg, P = 1.5 deg,
    GP2:
        UF : 1, UT : 2,
       J1 = 0.0 deg, J2 = 0.0 deg
 };
P[215] {
    GP1:
        UF : 6, UT : 5,     CONFIG: 'N U T, 0, 0, 0',
       X = -423.8 mm, Y = 518.4 mm, Z = 657.7 mm,
       W = 1.1 deg, P = 1.4 deg,
    GP2:
        UF : 1, UT : 2,
       J1 = 0.0 deg, J2 = 0.0 deg
 };
P[460] {
    GP1:
        UF : 6, UT : 5,     CONFIG: 'N U T, 0, 0, 0',
 X = -406.8 mm, Y = 589.4 mm, Z = 657.7 mm,       W = 1.1 deg, P = 1.4 deg,
    GP2:
        UF : 1, UT : 2,
       J1 = 0.0 deg, J2 = 0.0 deg
 };
P[216] {
    GP1:
        UF : 6, UT : 5,     CONFIG: 'N U T, 0, 0, 0',
       X = -432.5 mm, Y = 522.9 mm, Z = 657.7 mm,
       W = 1.0 deg, P = 1.1 deg,
    GP2:
        UF : 1, UT : 2,
       J1 = 0.0 deg, J2 = 0.0 deg
 };
P[461] {
    GP1:
        UF : 6, UT : 5,     CONFIG: 'N U T, 0, 0, 0',
 X = -415.5 mm, Y = 593.9 mm, Z = 657.7 mm,       W = 1.0 deg, P = 1.1 deg,
    GP2:
        UF : 1, UT : 2,
       J1 = 0.0 deg, J2 = 0.0 deg
 };
P[217] {
    GP1:
        UF : 6, UT : 5,     CONFIG: 'N U T, 0, 0, 0',
       X = -438.9 mm, Y = 526.1 mm, Z = 657.7 mm,
       W = 0.8 deg, P = 1.0 deg,
    GP2:
        UF : 1, UT : 2,
       J1 = 0.0 deg, J2 = 0.0 deg
 };
P[462] {
    GP1:
        UF : 6, UT : 5,     CONFIG: 'N U T, 0, 0, 0',
 X = -421.9 mm, Y = 597.1 mm, Z = 657.7 mm,       W = 0.8 deg, P = 1.0 deg,
    GP2:
        UF : 1, UT : 2,
       J1 = 0.0 deg, J2 = 0.0 deg
 };
P[218] {
    GP1:
        UF : 6, UT : 5,     CONFIG: 'N U T, 0, 0, 0',
       X = -440.9 mm, Y = 527.3 mm, Z = 657.7 mm,
       W = 0.8 deg, P = 0.9 deg,
    GP2:
        UF : 1, UT : 2,
       J1 = 0.0 deg, J2 = 0.0 deg
 };
P[463] {
    GP1:
        UF : 6, UT : 5,     CONFIG: 'N U T, 0, 0, 0',
 X = -423.9 mm, Y = 598.3 mm, Z = 657.7 mm,       W = 0.8 deg, P = 0.9 deg,
    GP2:
        UF : 1, UT : 2,
       J1 = 0.0 deg, J2 = 0.0 deg
 };
P[219] {
    GP1:
        UF : 6, UT : 5,     CONFIG: 'N U T, 0, 0, 0',
       X = -442.6 mm, Y = 528.8 mm, Z = 657.7 mm,
       W = 0.7 deg, P = 0.9 deg,
    GP2:
        UF : 1, UT : 2,
       J1 = 0.0 deg, J2 = 0.0 deg
 };
P[464] {
    GP1:
        UF : 6, UT : 5,     CONFIG: 'N U T, 0, 0, 0',
 X = -425.6 mm, Y = 599.8 mm, Z = 657.7 mm,       W = 0.7 deg, P = 0.9 deg,
    GP2:
        UF : 1, UT : 2,
       J1 = 0.0 deg, J2 = 0.0 deg
 };
P[220] {
    GP1:
        UF : 6, UT : 5,     CONFIG: 'N U T, 0, 0, 0',
       X = -444.1 mm, Y = 530.4 mm, Z = 657.7 mm,
       W = 0.7 deg, P = 0.9 deg,
    GP2:
        UF : 1, UT : 2,
       J1 = 0.0 deg, J2 = 0.0 deg
 };
P[465] {
    GP1:
        UF : 6, UT : 5,     CONFIG: 'N U T, 0, 0, 0',
 X = -427.1 mm, Y = 601.4 mm, Z = 657.7 mm,       W = 0.7 deg, P = 0.9 deg,
    GP2:
        UF : 1, UT : 2,
       J1 = 0.0 deg, J2 = 0.0 deg
 };
P[221] {
    GP1:
        UF : 6, UT : 5,     CONFIG: 'N U T, 0, 0, 0',
       X = -445.1 mm, Y = 531.7 mm, Z = 657.7 mm,
       W = 0.7 deg, P = 0.8 deg,
    GP2:
        UF : 1, UT : 2,
       J1 = 0.0 deg, J2 = 0.0 deg
 };
P[466] {
    GP1:
        UF : 6, UT : 5,     CONFIG: 'N U T, 0, 0, 0',
 X = -428.1 mm, Y = 602.7 mm, Z = 657.7 mm,       W = 0.7 deg, P = 0.8 deg,
    GP2:
        UF : 1, UT : 2,
       J1 = 0.0 deg, J2 = 0.0 deg
 };
P[222] {
    GP1:
        UF : 6, UT : 5,     CONFIG: 'N U T, 0, 0, 0',
       X = -450.0 mm, Y = 539.7 mm, Z = 657.7 mm,
       W = 0.5 deg, P = 0.6 deg,
    GP2:
        UF : 1, UT : 2,
       J1 = 0.0 deg, J2 = 0.0 deg
 };
P[467] {
    GP1:
        UF : 6, UT : 5,     CONFIG: 'N U T, 0, 0, 0',
 X = -433.0 mm, Y = 610.7 mm, Z = 657.7 mm,       W = 0.5 deg, P = 0.6 deg,
    GP2:
        UF : 1, UT : 2,
       J1 = 0.0 deg, J2 = 0.0 deg
 };
P[223] {
    GP1:
        UF : 6, UT : 5,     CONFIG: 'N U T, 0, 0, 0',
       X = -454.8 mm, Y = 547.8 mm, Z = 657.7 mm,
       W = 0.3 deg, P = 0.4 deg,
    GP2:
        UF : 1, UT : 2,
       J1 = 0.0 deg, J2 = 0.0 deg
 };
P[468] {
    GP1:
        UF : 6, UT : 5,     CONFIG: 'N U T, 0, 0, 0',
 X = -437.8 mm, Y = 618.8 mm, Z = 657.7 mm,       W = 0.3 deg, P = 0.4 deg,
    GP2:
        UF : 1, UT : 2,
       J1 = 0.0 deg, J2 = 0.0 deg
 };
P[224] {
    GP1:
        UF : 6, UT : 5,     CONFIG: 'N U T, 0, 0, 0',
       X = -456.7 mm, Y = 551.0 mm, Z = 657.7 mm,
       W = 0.3 deg, P = 0.3 deg,
    GP2:
        UF : 1, UT : 2,
       J1 = 0.0 deg, J2 = 0.0 deg
 };
P[469] {
    GP1:
        UF : 6, UT : 5,     CONFIG: 'N U T, 0, 0, 0',
 X = -439.7 mm, Y = 622.0 mm, Z = 657.7 mm,       W = 0.3 deg, P = 0.3 deg,
    GP2:
        UF : 1, UT : 2,
       J1 = 0.0 deg, J2 = 0.0 deg
 };
P[225] {
    GP1:
        UF : 6, UT : 5,     CONFIG: 'N U T, 0, 0, 0',
       X = -457.6 mm, Y = 552.7 mm, Z = 657.7 mm,
       W = 0.2 deg, P = 0.3 deg,
    GP2:
        UF : 1, UT : 2,
       J1 = 0.0 deg, J2 = 0.0 deg
 };
P[470] {
    GP1:
        UF : 6, UT : 5,     CONFIG: 'N U T, 0, 0, 0',
 X = -440.6 mm, Y = 623.7 mm, Z = 657.7 mm,       W = 0.2 deg, P = 0.3 deg,
    GP2:
        UF : 1, UT : 2,
       J1 = 0.0 deg, J2 = 0.0 deg
 };
P[226] {
    GP1:
        UF : 6, UT : 5,     CONFIG: 'N U T, 0, 0, 0',
       X = -458.1 mm, Y = 554.0 mm, Z = 657.7 mm,
       W = 0.2 deg, P = 0.2 deg,
    GP2:
        UF : 1, UT : 2,
       J1 = 0.0 deg, J2 = 0.0 deg
 };
P[471] {
    GP1:
        UF : 6, UT : 5,     CONFIG: 'N U T, 0, 0, 0',
 X = -441.1 mm, Y = 625.0 mm, Z = 657.7 mm,       W = 0.2 deg, P = 0.2 deg,
    GP2:
        UF : 1, UT : 2,
       J1 = 0.0 deg, J2 = 0.0 deg
 };
P[227] {
    GP1:
        UF : 6, UT : 5,     CONFIG: 'N U T, 0, 0, 0',
       X = -458.3 mm, Y = 555.3 mm, Z = 657.7 mm,
       W = 0.2 deg, P = 0.2 deg,
    GP2:
        UF : 1, UT : 2,
       J1 = 0.0 deg, J2 = 0.0 deg
 };
P[472] {
    GP1:
        UF : 6, UT : 5,     CONFIG: 'N U T, 0, 0, 0',
 X = -441.3 mm, Y = 626.3 mm, Z = 657.7 mm,       W = 0.2 deg, P = 0.2 deg,
    GP2:
        UF : 1, UT : 2,
       J1 = 0.0 deg, J2 = 0.0 deg
 };
P[228] {
    GP1:
        UF : 6, UT : 5,     CONFIG: 'N U T, 0, 0, 0',
       X = -458.3 mm, Y = 555.9 mm, Z = 657.7 mm,
       W = 0.2 deg, P = 0.2 deg,
    GP2:
        UF : 1, UT : 2,
       J1 = 0.0 deg, J2 = 0.0 deg
 };
P[473] {
    GP1:
        UF : 6, UT : 5,     CONFIG: 'N U T, 0, 0, 0',
 X = -441.3 mm, Y = 626.9 mm, Z = 657.7 mm,       W = 0.2 deg, P = 0.2 deg,
    GP2:
        UF : 1, UT : 2,
       J1 = 0.0 deg, J2 = 0.0 deg
 };
P[229] {
    GP1:
        UF : 6, UT : 5,     CONFIG: 'N U T, 0, 0, 0',
       X = -458.2 mm, Y = 557.1 mm, Z = 657.7 mm,
       W = 0.1 deg, P = 0.2 deg,
    GP2:
        UF : 1, UT : 2,
       J1 = 0.0 deg, J2 = 0.0 deg
 };
P[474] {
    GP1:
        UF : 6, UT : 5,     CONFIG: 'N U T, 0, 0, 0',
 X = -441.2 mm, Y = 628.1 mm, Z = 657.7 mm,       W = 0.1 deg, P = 0.2 deg,
    GP2:
        UF : 1, UT : 2,
       J1 = 0.0 deg, J2 = 0.0 deg
 };
P[230] {
    GP1:
        UF : 6, UT : 5,     CONFIG: 'N U T, 0, 0, 0',
       X = -458.1 mm, Y = 558.0 mm, Z = 657.7 mm,
       W = 0.1 deg, P = 0.2 deg,
    GP2:
        UF : 1, UT : 2,
       J1 = 0.0 deg, J2 = 0.0 deg
 };
P[475] {
    GP1:
        UF : 6, UT : 5,     CONFIG: 'N U T, 0, 0, 0',
 X = -441.1 mm, Y = 629.0 mm, Z = 657.7 mm,       W = 0.1 deg, P = 0.2 deg,
    GP2:
        UF : 1, UT : 2,
       J1 = 0.0 deg, J2 = 0.0 deg
 };
P[231] {
    GP1:
        UF : 6, UT : 5,     CONFIG: 'N U T, 0, 0, 0',
       X = -457.8 mm, Y = 558.6 mm, Z = 657.7 mm,
       W = 0.1 deg, P = 0.1 deg,
    GP2:
        UF : 1, UT : 2,
       J1 = 0.0 deg, J2 = 0.0 deg
 };
P[476] {
    GP1:
        UF : 6, UT : 5,     CONFIG: 'N U T, 0, 0, 0',
 X = -440.8 mm, Y = 629.6 mm, Z = 657.7 mm,       W = 0.1 deg, P = 0.1 deg,
    GP2:
        UF : 1, UT : 2,
       J1 = 0.0 deg, J2 = 0.0 deg
 };
P[232] {
    GP1:
        UF : 6, UT : 5,     CONFIG: 'N U T, 0, 0, 0',
       X = -457.2 mm, Y = 560.0 mm, Z = 657.7 mm,
       W = 0.1 deg, P = 0.1 deg,
    GP2:
        UF : 1, UT : 2,
       J1 = 0.0 deg, J2 = 0.0 deg
 };
P[477] {
    GP1:
        UF : 6, UT : 5,     CONFIG: 'N U T, 0, 0, 0',
 X = -440.2 mm, Y = 631.0 mm, Z = 657.7 mm,       W = 0.1 deg, P = 0.1 deg,
    GP2:
        UF : 1, UT : 2,
       J1 = 0.0 deg, J2 = 0.0 deg
 };
P[233] {
    GP1:
        UF : 6, UT : 5,     CONFIG: 'N U T, 0, 0, 0',
       X = -456.3 mm, Y = 561.3 mm, Z = 657.7 mm,
       W = 0.1 deg, P = 0.1 deg,
    GP2:
        UF : 1, UT : 2,
       J1 = 0.0 deg, J2 = 0.0 deg
 };
P[478] {
    GP1:
        UF : 6, UT : 5,     CONFIG: 'N U T, 0, 0, 0',
 X = -439.3 mm, Y = 632.3 mm, Z = 657.7 mm,       W = 0.1 deg, P = 0.1 deg,
    GP2:
        UF : 1, UT : 2,
       J1 = 0.0 deg, J2 = 0.0 deg
 };
P[234] {
    GP1:
        UF : 6, UT : 5,     CONFIG: 'N U T, 0, 0, 0',
       X = -455.2 mm, Y = 562.3 mm, Z = 657.7 mm,
       W = 0.0 deg, P = 0.1 deg,
    GP2:
        UF : 1, UT : 2,
       J1 = 0.0 deg, J2 = 0.0 deg
 };
P[479] {
    GP1:
        UF : 6, UT : 5,     CONFIG: 'N U T, 0, 0, 0',
 X = -438.2 mm, Y = 633.3 mm, Z = 657.7 mm,       W = 0.0 deg, P = 0.1 deg,
    GP2:
        UF : 1, UT : 2,
       J1 = 0.0 deg, J2 = 0.0 deg
 };
P[235] {
    GP1:
        UF : 6, UT : 5,     CONFIG: 'N U T, 0, 0, 0',
       X = -447.1 mm, Y = 567.6 mm, Z = 657.7 mm,
       W = 0.0 deg, P = 0.0 deg,
    GP2:
        UF : 1, UT : 2,
       J1 = 0.0 deg, J2 = 0.0 deg
 };
P[480] {
    GP1:
        UF : 6, UT : 5,     CONFIG: 'N U T, 0, 0, 0',
 X = -430.1 mm, Y = 638.6 mm, Z = 657.7 mm,       W = 0.0 deg, P = 0.0 deg,
    GP2:
        UF : 1, UT : 2,
       J1 = 0.0 deg, J2 = 0.0 deg
 };
P[236] {
    GP1:
        UF : 6, UT : 5,     CONFIG: 'N U T, 0, 0, 0',
       X = -439.0 mm, Y = 572.9 mm, Z = 657.7 mm,
       W = 0.0 deg, P = 0.0 deg,
    GP2:
        UF : 1, UT : 2,
       J1 = 0.0 deg, J2 = 0.0 deg
 };
P[481] {
    GP1:
        UF : 6, UT : 5,     CONFIG: 'N U T, 0, 0, 0',
 X = -422.0 mm, Y = 643.9 mm, Z = 657.7 mm,       W = 0.0 deg, P = 0.0 deg,
    GP2:
        UF : 1, UT : 2,
       J1 = 0.0 deg, J2 = 0.0 deg
 };
P[237] {
    GP1:
        UF : 6, UT : 5,     CONFIG: 'N U T, 0, 0, 0',
       X = -430.9 mm, Y = 578.1 mm, Z = 657.7 mm,
       W = 0.0 deg, P = 0.0 deg,
    GP2:
        UF : 1, UT : 2,
       J1 = 0.0 deg, J2 = 0.0 deg
 };
P[482] {
    GP1:
        UF : 6, UT : 5,     CONFIG: 'N U T, 0, 0, 0',
 X = -413.9 mm, Y = 649.1 mm, Z = 657.7 mm,       W = 0.0 deg, P = 0.0 deg,
    GP2:
        UF : 1, UT : 2,
       J1 = 0.0 deg, J2 = 0.0 deg
 };
P[238] {
    GP1:
        UF : 6, UT : 5,     CONFIG: 'N U T, 0, 0, 0',
       X = -422.8 mm, Y = 583.4 mm, Z = 657.7 mm,
       W = 0.0 deg, P = 0.0 deg,
    GP2:
        UF : 1, UT : 2,
       J1 = 0.0 deg, J2 = 0.0 deg
 };
P[483] {
    GP1:
        UF : 6, UT : 5,     CONFIG: 'N U T, 0, 0, 0',
 X = -405.8 mm, Y = 654.4 mm, Z = 657.7 mm,       W = 0.0 deg, P = 0.0 deg,
    GP2:
        UF : 1, UT : 2,
       J1 = 0.0 deg, J2 = 0.0 deg
 };
P[239] {
    GP1:
        UF : 6, UT : 5,     CONFIG: 'N U T, 0, 0, 0',
       X = -414.8 mm, Y = 588.6 mm, Z = 657.7 mm,
       W = 0.0 deg, P = 0.0 deg,
    GP2:
        UF : 1, UT : 2,
       J1 = 0.0 deg, J2 = 0.0 deg
 };
P[484] {
    GP1:
        UF : 6, UT : 5,     CONFIG: 'N U T, 0, 0, 0',
 X = -397.8 mm, Y = 659.6 mm, Z = 657.7 mm,       W = 0.0 deg, P = 0.0 deg,
    GP2:
        UF : 1, UT : 2,
       J1 = 0.0 deg, J2 = 0.0 deg
 };
P[240] {
    GP1:
        UF : 6, UT : 5,     CONFIG: 'N U T, 0, 0, 0',
       X = -406.7 mm, Y = 593.9 mm, Z = 657.7 mm,
       W = 0.0 deg, P = 0.0 deg,
    GP2:
        UF : 1, UT : 2,
       J1 = 0.0 deg, J2 = 0.0 deg
 };
P[485] {
    GP1:
        UF : 6, UT : 5,     CONFIG: 'N U T, 0, 0, 0',
 X = -389.7 mm, Y = 664.9 mm, Z = 657.7 mm,       W = 0.0 deg, P = 0.0 deg,
    GP2:
        UF : 1, UT : 2,
       J1 = 0.0 deg, J2 = 0.0 deg
 };
P[241] {
    GP1:
        UF : 6, UT : 5,     CONFIG: 'N U T, 0, 0, 0',
       X = -398.6 mm, Y = 599.1 mm, Z = 657.7 mm,
       W = 0.0 deg, P = 0.0 deg,
    GP2:
        UF : 1, UT : 2,
       J1 = 0.0 deg, J2 = 0.0 deg
 };
P[486] {
    GP1:
        UF : 6, UT : 5,     CONFIG: 'N U T, 0, 0, 0',
 X = -381.6 mm, Y = 670.1 mm, Z = 657.7 mm,       W = 0.0 deg, P = 0.0 deg,
    GP2:
        UF : 1, UT : 2,
       J1 = 0.0 deg, J2 = 0.0 deg
 };
P[242] {
    GP1:
        UF : 6, UT : 5,     CONFIG: 'N U T, 0, 0, 0',
       X = -390.5 mm, Y = 604.3 mm, Z = 657.7 mm,
       W = 0.0 deg, P = 0.0 deg,
    GP2:
        UF : 1, UT : 2,
       J1 = 0.0 deg, J2 = 0.0 deg
 };
P[487] {
    GP1:
        UF : 6, UT : 5,     CONFIG: 'N U T, 0, 0, 0',
 X = -373.5 mm, Y = 675.3 mm, Z = 657.7 mm,       W = 0.0 deg, P = 0.0 deg,
    GP2:
        UF : 1, UT : 2,
       J1 = 0.0 deg, J2 = 0.0 deg
 };
P[243] {
    GP1:
        UF : 6, UT : 5,     CONFIG: 'N U T, 0, 0, 0',
       X = -382.5 mm, Y = 609.6 mm, Z = 657.7 mm,
       W = 0.0 deg, P = 0.0 deg,
    GP2:
        UF : 1, UT : 2,
       J1 = 0.0 deg, J2 = 0.0 deg
 };
P[488] {
    GP1:
        UF : 6, UT : 5,     CONFIG: 'N U T, 0, 0, 0',
 X = -365.5 mm, Y = 680.6 mm, Z = 657.7 mm,       W = 0.0 deg, P = 0.0 deg,
    GP2:
        UF : 1, UT : 2,
       J1 = 0.0 deg, J2 = 0.0 deg
 };
/END
